(* PLC project lng-production, Generated TextualNotationConverter 1.0 *)
(* stored: creationDateTime 2025-07-30T12:00:00, modificationDateTime 2025-01-30T12:00:00 *)

FUNCTION_BLOCK ANALOG_IN
  VAR_INPUT
    Name : STRING;
    Description : STRING;
    Raw_Signal : REAL;
    PV_High : REAL;
    PV_Low : REAL;
    Scaling_Slope : REAL;
    Scaling_Offset : REAL;
    Alarm_Enable : BOOL;
  END_VAR
  VAR_OUTPUT
    PV : REAL;
    High_Alarm : BOOL;
    Low_Alarm : BOOL;
    General_Fault : BOOL;
  END_VAR

            
          
END_FUNCTION_BLOCK

FUNCTION_BLOCK RATIO_CONTROL
  VAR_INPUT
    Name : STRING;
    Description : STRING;
    Auto : BOOL;
    PrimaryPV : REAL;
    SecondaryPV : REAL;
    RatioSP : REAL;
    Bias : REAL;
    TrimKp : REAL;
    TrimTi : STRING;
    MV_MIN : REAL;
    MV_MAX : REAL;
    ManOut : REAL;
    Inhibit : BOOL;
  END_VAR
  VAR_OUTPUT
    SlaveSP : REAL;
    ActiveRatio : REAL;
    RatioErr : REAL;
  END_VAR

            
          
END_FUNCTION_BLOCK

FUNCTION_BLOCK VALVE_ELECTRIC
  VAR_INPUT
    Name : STRING;
    Description : STRING;
    Control_Signal : REAL;
    Manual_Mode : BOOL;
    Manual_Position : REAL;
    Open_Limit : REAL;
    Close_Limit : REAL;
    Timeout : STRING;
    Inhibit : BOOL;
  END_VAR
  VAR_OUTPUT
    Valve_Position : REAL;
    Feedback_Pos : REAL;
    Valve_Moving : BOOL;
    Position_Error : BOOL;
    Alarm : BOOL;
  END_VAR

            
          
END_FUNCTION_BLOCK

PROGRAM Section2
  VAR
    FT101_FeedGasFlow_PV : REAL;
    IT102_LiqSepFlow_PV : REAL;
    LT101_SlugCatcherLevel_PV : REAL;
    DP101_InletSepDP_PV : REAL;
    DP102_InletSepDP_PV : REAL;
    IIC101_LiqSepFlow_SP : REAL;
    IIC101_CalculatedRatio : REAL;
  END_VAR
  VAR
    DP-101 : ANALOG_IN;
    DP-102 : ANALOG_IN;
    FT-101 : ANALOG_IN;
    IT-102 : ANALOG_IN;
    LT-101 : ANALOG_IN;
    IIC-101 : RATIO_CONTROL;
    LCV-101 : VALVE_ELECTRIC;
  END_VAR

(* FBD diagram, written out as Structured Text *)
DP-101(PV_High := 10, PV_Low := 0, Alarm_Enable := TRUE, Scaling_Slope := 0.625, Scaling_Offset := -2.5);
DP101_InletSepDP_PV := DP-101.PV;
DP-102(PV_High := 10, PV_Low := 0, Alarm_Enable := TRUE, Scaling_Slope := 0.625, Scaling_Offset := -2.5);
DP102_InletSepDP_PV := DP-102.PV;
FT-101(PV_High := 5000, PV_Low := 100, Alarm_Enable := TRUE, Scaling_Slope := 312.5, Scaling_Offset := -1250);
FT101_FeedGasFlow_PV := FT-101.PV;
IT-102(PV_High := 2000, PV_Low := 0, Alarm_Enable := TRUE, Scaling_Slope := 125, Scaling_Offset := -500);
LT-101(PV_High := 80, PV_Low := 0, Alarm_Enable := TRUE, Scaling_Slope := 6.25, Scaling_Offset := -25);
IIC-101(PrimaryPV := FT-101.PV, SecondaryPV := IT-102.PV, Inhibit := DP-101.High_Alarm OR DP-102.High_Alarm OR LT-101.High_Alarm OR FT-101.Low_Alarm, Auto := TRUE, RatioSP := 2.5, Bias := 0, MV_MIN := 0, MV_MAX := 2000, ManOut := 500);
IIC101_CalculatedRatio := IIC-101.ActiveRatio;
IIC101_LiqSepFlow_SP := IIC-101.SlaveSP;
IT102_LiqSepFlow_PV := IT-102.PV;
LT101_SlugCatcherLevel_PV := LT-101.PV;
LCV-101(Control_Signal := IIC-101.SlaveSP, Inhibit := IT-102.High_Alarm OR IT-102.Low_Alarm OR FT-101.Low_Alarm OR IT-102.General_Fault, Manual_Mode := FALSE, Manual_Position := 0, Open_Limit := 100, Close_Limit := 0);
END_PROGRAM

FUNCTION_BLOCK BOOL_IN
  VAR_INPUT
    Name : STRING;
    Description : STRING;
    Bool_In : BOOL;
    Alarm_OnTrue : BOOL;
    Alarm_OnFalse : BOOL;
    Latch_Enable : BOOL;
    Reset_Latch : BOOL;
  END_VAR
  VAR_OUTPUT
    Bool_Out : BOOL;
    Alarm_Active : BOOL;
    Latched_Status : BOOL;
  END_VAR

            
          
END_FUNCTION_BLOCK

FUNCTION_BLOCK DIGITAL_IN
  VAR_INPUT
    Name : STRING;
    Description : STRING;
    DI_Raw : BOOL;
    DebounceTime : STRING;
    EnableAlarm : BOOL;
  END_VAR
  VAR_OUTPUT
    DI_Out : BOOL;
    Fault_State : BOOL;
  END_VAR

            
          
END_FUNCTION_BLOCK

FUNCTION_BLOCK DUTY_STANDBY
  VAR_INPUT
    Name : STRING;
    Description : STRING;
    Enable : BOOL;
    StartRequest : BOOL;
    AlternateEnable : BOOL;
    ForcePumpA : BOOL;
    ForcePumpB : BOOL;
    DutyElapsed : BOOL;
    MinRunElapsed : BOOL;
    SwitchoverDelayElapsed : BOOL;
    StartTimeoutElapsed : BOOL;
    PumpA_RunFB : BOOL;
    PumpB_RunFB : BOOL;
    PumpA_Fault : BOOL;
    PumpB_Fault : BOOL;
    Reset : BOOL;
    Inhibit : BOOL;
  END_VAR
  VAR_OUTPUT
    CmdPumpA : BOOL;
    CmdPumpB : BOOL;
    ActiveIsA : BOOL;
    SwitchedDueToDuty : BOOL;
    SwitchedDueToFailure : BOOL;
    Alarm_FailedStart_A : BOOL;
    Alarm_FailedStart_B : BOOL;
    Alarm_NoAvailablePump : BOOL;
  END_VAR

            
          
END_FUNCTION_BLOCK

FUNCTION_BLOCK MOTOR_2SPD
  VAR_INPUT
    Name : STRING;
    Description : STRING;
    Start_Cmd : BOOL;
    Stop_Cmd : BOOL;
    Speed_High_Cmd : BOOL;
    Speed_Low_Cmd : BOOL;
    Inhibit : BOOL;
  END_VAR
  VAR_OUTPUT
    Motor_Start_Out : BOOL;
    FB_Running : BOOL;
    FB_Trip : BOOL;
    FB_HighSpeed : BOOL;
    FB_LowSpeed : BOOL;
    Alarm_Speed_Error : BOOL;
  END_VAR

            
          
END_FUNCTION_BLOCK

FUNCTION_BLOCK MOTOR_ON_OFF
  VAR_INPUT
    Name : STRING;
    Description : STRING;
    Start_Cmd : BOOL;
    Stop_Cmd : BOOL;
    Start_Delay : STRING;
    MinRunTime : STRING;
    Inhibit : BOOL;
  END_VAR
  VAR_OUTPUT
    Motor_Start_Out : BOOL;
    FB_Running : BOOL;
    FB_Trip : BOOL;
    Alarm_Start_Fail : BOOL;
    Alarm_Stop_Fail : BOOL;
  END_VAR

            
          
END_FUNCTION_BLOCK

FUNCTION_BLOCK MOTOR_VSD
  VAR_INPUT
    Name : STRING;
    Description : STRING;
    Start_Cmd : BOOL;
    Stop_Cmd : BOOL;
    Speed_SP : REAL;
    Accel_Ramp : STRING;
    Decel_Ramp : STRING;
    Inhibit : BOOL;
  END_VAR
  VAR_OUTPUT
    Speed_Out : REAL;
    FB_Running : BOOL;
    FB_Fault : BOOL;
    FB_Ready : BOOL;
    FB_ActualSpeed : REAL;
    Alarm_Speed_Deviation : BOOL;
    Alarm_Comm_Fail : BOOL;
  END_VAR

            
          
END_FUNCTION_BLOCK

FUNCTION_BLOCK PID_BASIC
  VAR_INPUT
    Name : STRING;
    Description : STRING;
    AUTO : BOOL;
    PV : REAL;
    SP : REAL;
    MV_MIN : REAL;
    MV_MAX : REAL;
    X0 : REAL;
    KP : REAL;
    TR : REAL;
    TD : REAL;
    PV_High : REAL;
    PV_Low : REAL;
    Deviation_Limit : REAL;
    Inhibit : BOOL;
  END_VAR
  VAR_OUTPUT
    PV_High_Alarm : BOOL;
    PV_Low_Alarm : BOOL;
    Deviation_Alarm : BOOL;
    XOUT : REAL;
  END_VAR

            
          
END_FUNCTION_BLOCK

FUNCTION_BLOCK SPLIT_RANGE
  VAR_INPUT
    Name : STRING;
    Description : STRING;
    IN : REAL;
    Split_Point : REAL;
    Output1_Start : REAL;
    Output1_End : REAL;
    Output2_Start : REAL;
    Output2_End : REAL;
  END_VAR
  VAR_OUTPUT
    OUT1 : REAL;
    OUT2 : REAL;
  END_VAR

            
          
END_FUNCTION_BLOCK

FUNCTION_BLOCK VALVE_ON_OFF
  VAR_INPUT
    Name : STRING;
    Description : STRING;
    Open_Cmd : BOOL;
    Close_Cmd : BOOL;
    Timeout : STRING;
    Inhibit : BOOL;
  END_VAR
  VAR_OUTPUT
    FB_Opened : BOOL;
    FB_Closed : BOOL;
    Valve_Open_Out : BOOL;
    Valve_Close_Out : BOOL;
    Alarm_Position_Error : BOOL;
    Alarm_General : BOOL;
  END_VAR

            
          
END_FUNCTION_BLOCK

FUNCTION_BLOCK VOTING_ANALOG
  VAR_INPUT
    Name : STRING;
    Description : STRING;
    Input1 : REAL;
    Input2 : REAL;
    Input3 : REAL;
    Deviation_Limit : REAL;
    Voting_Scheme : STRING;
    EnableAlarm : BOOL;
    Inhibit : BOOL;
  END_VAR
  VAR_OUTPUT
    Voted_Output : REAL;
    Sensor1_Fault : BOOL;
    Sensor2_Fault : BOOL;
    Sensor3_Fault : BOOL;
    Alarm_Voting_Error : BOOL;
    Healthy_Sensors_Count : INT;
  END_VAR

            
          
END_FUNCTION_BLOCK

PROGRAM Section3
  VAR
    TT201_Temperature_PV : REAL;
    TIC201_Output_MV_Pct : REAL;
    PT201_Pressure_PV : REAL;
    LT201_Level_PV : REAL;
    AI201_CO2_PV : REAL;
  END_VAR
  VAR
    AI-201 : ANALOG_IN;
    FV-101 : VALVE_ELECTRIC;
    LT-201 : ANALOG_IN;
    PT-201 : ANALOG_IN;
    TIC-201 : PID_BASIC;
    TT-201 : ANALOG_IN;
  END_VAR
  VAR  (* added by the conversion: wires and edge detectors of the diagram *)
    _OR56_OUT : BOOL;
  END_VAR

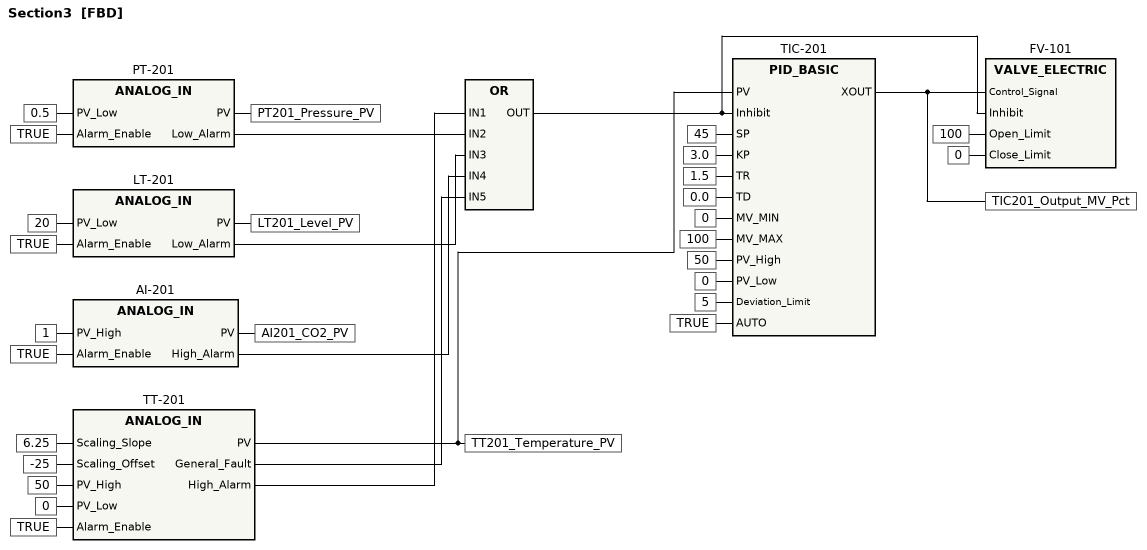
(* FBD diagram, written out as Structured Text *)
AI-201(PV_High := 1, Alarm_Enable := TRUE);
AI201_CO2_PV := AI-201.PV;
LT-201(PV_Low := 20, Alarm_Enable := TRUE);
LT201_Level_PV := LT-201.PV;
PT-201(PV_Low := 0.5, Alarm_Enable := TRUE);
PT201_Pressure_PV := PT-201.PV;
TT-201(Scaling_Slope := 6.25, Scaling_Offset := -25, PV_High := 50, PV_Low := 0, Alarm_Enable := TRUE);
_OR56_OUT := TT-201.High_Alarm OR PT-201.Low_Alarm OR LT-201.Low_Alarm OR AI-201.High_Alarm OR TT-201.General_Fault;
TIC-201(PV := TT-201.PV, Inhibit := _OR56_OUT, SP := 45, KP := 3.0, TR := 1.5, TD := 0.0, MV_MIN := 0, MV_MAX := 100, PV_High := 50, PV_Low := 0, Deviation_Limit := 5, AUTO := TRUE);
TIC201_Output_MV_Pct := TIC-201.XOUT;
TT201_Temperature_PV := TT-201.PV;
FV-101(Control_Signal := TIC-201.XOUT, Inhibit := _OR56_OUT, Open_Limit := 100, Close_Limit := 0);
END_PROGRAM

PROGRAM Section4
  VAR
    FT301_FeedGasFlow_PV : REAL;
    AI302_Mercury_PV : REAL;
    AI303_Mercury_PV : REAL;
    AI304_OutletH2O_PV : REAL;
    DP301_BedDP_PV : REAL;
    FFIC303_RegenGasFlow_SP : REAL;
  END_VAR
  VAR
    AI-302 : ANALOG_IN;
    AI-303 : ANALOG_IN;
    AI-304 : ANALOG_IN;
    DI-301 : DIGITAL_IN;
    DP-301 : ANALOG_IN;
    FIC-302 : PID_BASIC;
    FT-301 : ANALOG_IN;
    FV-302 : VALVE_ELECTRIC;
    FFIC-303 : RATIO_CONTROL;
  END_VAR
  VAR  (* added by the conversion: wires and edge detectors of the diagram *)
    _OR91_OUT : BOOL;
  END_VAR

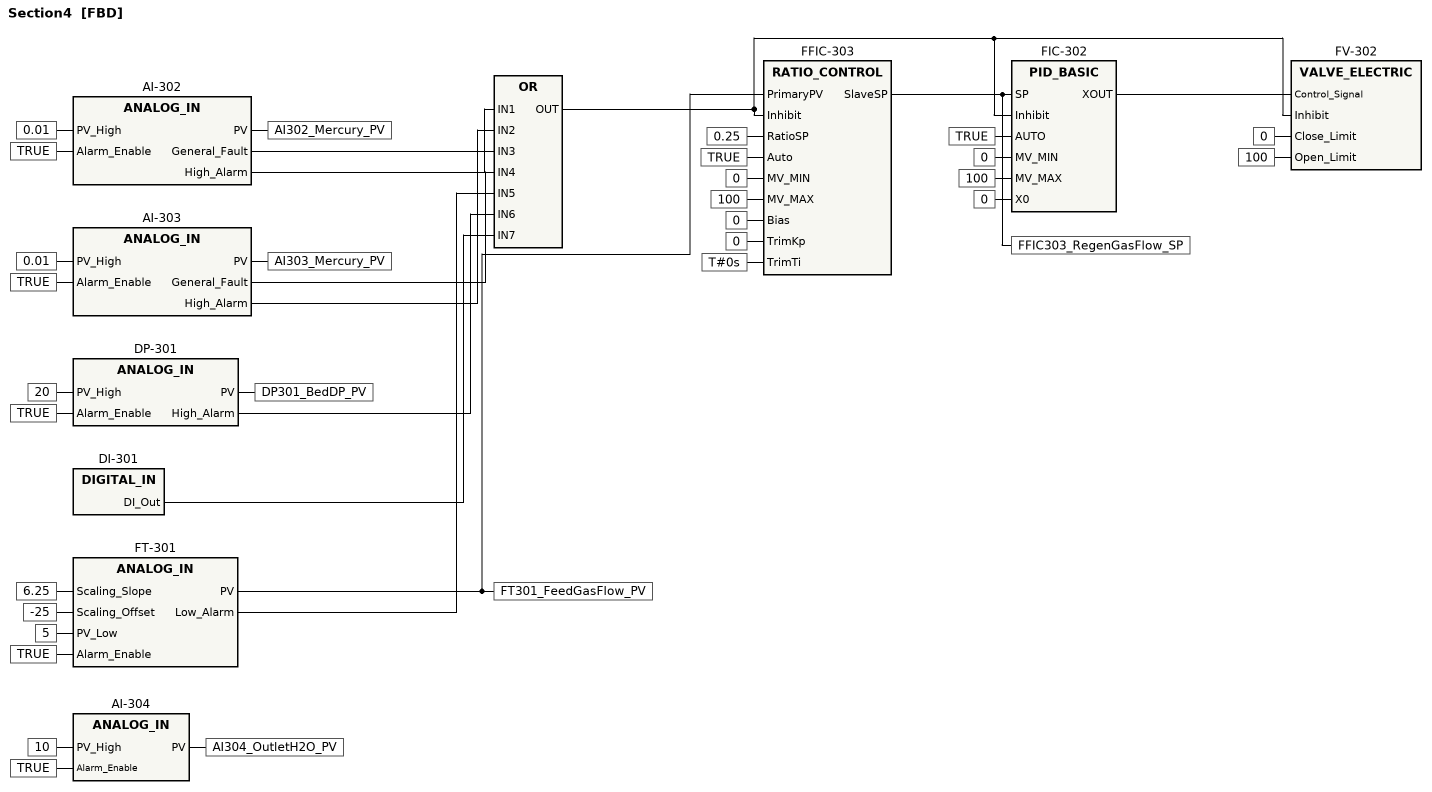
(* FBD diagram, written out as Structured Text *)
AI-302(PV_High := 0.01, Alarm_Enable := TRUE);
AI302_Mercury_PV := AI-302.PV;
AI-303(PV_High := 0.01, Alarm_Enable := TRUE);
AI303_Mercury_PV := AI-303.PV;
AI-304(PV_High := 10, Alarm_Enable := TRUE);
AI304_OutletH2O_PV := AI-304.PV;
DP-301(PV_High := 20, Alarm_Enable := TRUE);
DP301_BedDP_PV := DP-301.PV;
FT-301(Scaling_Slope := 6.25, Scaling_Offset := -25, PV_Low := 5, Alarm_Enable := TRUE);
DI-301();
_OR91_OUT := AI-302.High_Alarm OR AI-303.High_Alarm OR AI-302.General_Fault OR AI-303.General_Fault OR FT-301.Low_Alarm OR DP-301.High_Alarm OR DI-301.DI_Out;
FFIC-303(PrimaryPV := FT-301.PV, Inhibit := _OR91_OUT, RatioSP := 0.25, Auto := TRUE, MV_MIN := 0, MV_MAX := 100, Bias := 0, TrimKp := 0, TrimTi := T#0s);
FFIC303_RegenGasFlow_SP := FFIC-303.SlaveSP;
FT301_FeedGasFlow_PV := FT-301.PV;
FIC-302(SP := FFIC-303.SlaveSP, Inhibit := _OR91_OUT, AUTO := TRUE, MV_MIN := 0, MV_MAX := 100, X0 := 0);
FV-302(Control_Signal := FIC-302.XOUT, Inhibit := _OR91_OUT, Close_Limit := 0, Open_Limit := 100);
END_PROGRAM

PROGRAM Section5
  VAR
    PT_401_Pressure_PV : REAL;
    PT_401A_Pressure_PV : REAL;
    PT_401B_Pressure_PV : REAL;
    PT_401C_Pressure_PV : REAL;
    TT_105_Temperature_PV : REAL;
    TT_106_Temperature_PV : REAL;
    TT_107_Temperature_PV : REAL;
    FA_401_Flow_PV : REAL;
    FA_402A_Flow_PV : REAL;
    FA_402B_Flow_PV : REAL;
    FA_402C_Flow_PV : REAL;
    PVT_401_VotedPressure : REAL;
    TVT_402_VotedTemperature : REAL;
    PVT_401_Healthy_Count : INT;
    DA_401A_Deviation : BOOL;
    DA_401B_Deviation : BOOL;
    DA_401C_Deviation : BOOL;
    DA_402A_Deviation : BOOL;
    DA_402B_Deviation : BOOL;
    DA_402C_Deviation : BOOL;
    DA_402_Degraded : BOOL;
    MA_401_Alarm : BOOL;
  END_VAR
  VAR
    PT-401 : ANALOG_IN;
    PT-401A : ANALOG_IN;
    PT-401B : ANALOG_IN;
    PT-401C : ANALOG_IN;
    TT-105 : ANALOG_IN;
    TT-106 : ANALOG_IN;
    TT-107 : ANALOG_IN;
    FA-401 : ANALOG_IN;
    FA-402A : ANALOG_IN;
    FA-402B : ANALOG_IN;
    FA-402C : ANALOG_IN;
    PVT-401 : VOTING_ANALOG;
    TVT-402 : VOTING_ANALOG;
    PV-102_Control : PID_BASIC;
    PV-102 : VALVE_ELECTRIC;
    FV-107 : VALVE_ELECTRIC;
    XV-104 : VALVE_ON_OFF;
  END_VAR
  VAR  (* added by the conversion: wires and edge detectors of the diagram *)
    _MULT134_OUT : REAL;
    _OR155_OUT : BOOL;
    _AND132_OUT : BOOL;
    _OR156_OUT : BOOL;
  END_VAR

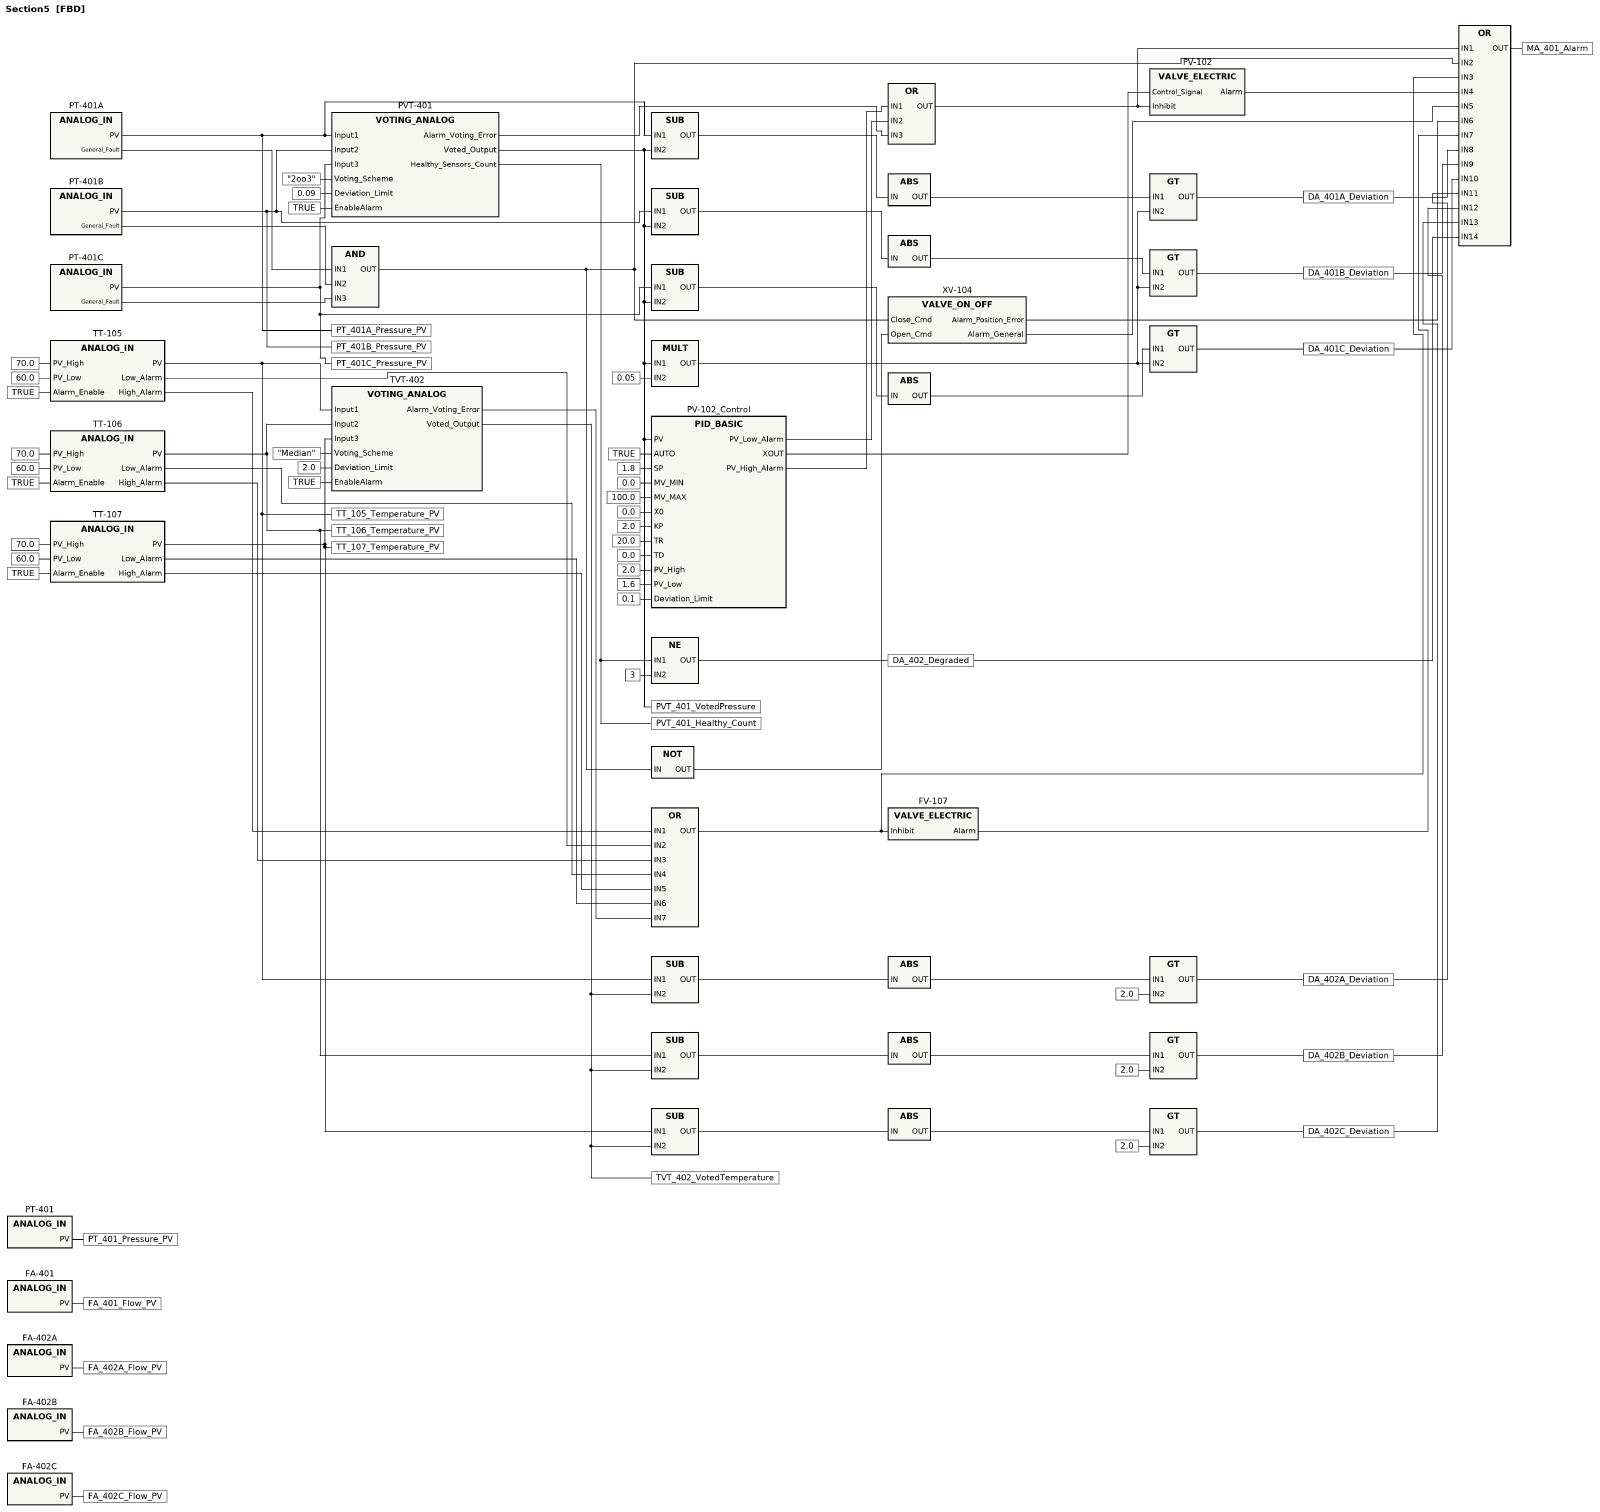
(* FBD diagram, written out as Structured Text *)
PT-401A();
PT-401B();
PT-401C();
PVT-401(Input1 := PT-401A.PV, Input2 := PT-401B.PV, Input3 := PT-401C.PV, Voting_Scheme := "2oo3", Deviation_Limit := 0.09, EnableAlarm := TRUE);
_MULT134_OUT := MULT(PVT-401.Voted_Output, 0.05);
DA_401A_Deviation := ABS(PT-401A.PV - PVT-401.Voted_Output) > _MULT134_OUT;
DA_401B_Deviation := ABS(PT-401B.PV - PVT-401.Voted_Output) > _MULT134_OUT;
DA_401C_Deviation := ABS(PT-401C.PV - PVT-401.Voted_Output) > _MULT134_OUT;
TT-105(PV_High := 70.0, PV_Low := 60.0, Alarm_Enable := TRUE);
TT-106(PV_High := 70.0, PV_Low := 60.0, Alarm_Enable := TRUE);
TT-107(PV_High := 70.0, PV_Low := 60.0, Alarm_Enable := TRUE);
TVT-402(Input1 := TT-105.PV, Input2 := TT-106.PV, Input3 := TT-107.PV, Voting_Scheme := "Median", Deviation_Limit := 2.0, EnableAlarm := TRUE);
DA_402A_Deviation := ABS(TT-105.PV - TVT-402.Voted_Output) > 2.0;
DA_402B_Deviation := ABS(TT-106.PV - TVT-402.Voted_Output) > 2.0;
DA_402C_Deviation := ABS(TT-107.PV - TVT-402.Voted_Output) > 2.0;
DA_402_Degraded := PVT-401.Healthy_Sensors_Count <> 3;
FA-401();
FA_401_Flow_PV := FA-401.PV;
FA-402A();
FA_402A_Flow_PV := FA-402A.PV;
FA-402B();
FA_402B_Flow_PV := FA-402B.PV;
FA-402C();
FA_402C_Flow_PV := FA-402C.PV;
PV-102_Control(PV := PVT-401.Voted_Output, AUTO := TRUE, SP := 1.8, MV_MIN := 0.0, MV_MAX := 100.0, X0 := 0.0, KP := 2.0, TR := 20.0, TD := 0.0, PV_High := 2.0, PV_Low := 1.6, Deviation_Limit := 0.1);
_OR155_OUT := PV-102_Control.PV_High_Alarm OR PV-102_Control.PV_Low_Alarm OR PVT-401.Alarm_Voting_Error;
_AND132_OUT := PT-401A.General_Fault AND PT-401B.General_Fault AND PT-401C.General_Fault;
_OR156_OUT := TT-105.High_Alarm OR TT-105.Low_Alarm OR TT-106.High_Alarm OR TT-106.Low_Alarm OR TT-107.High_Alarm OR TT-107.Low_Alarm OR TVT-402.Alarm_Voting_Error;
PV-102(Control_Signal := PV-102_Control.XOUT, Inhibit := _OR155_OUT);
XV-104(Close_Cmd := _AND132_OUT, Open_Cmd := NOT _AND132_OUT);
FV-107(Inhibit := _OR156_OUT);
MA_401_Alarm := _OR155_OUT OR _AND132_OUT OR _OR156_OUT OR PV-102.Alarm OR XV-104.Alarm_General OR XV-104.Alarm_Position_Error OR FV-107.Alarm OR ABS(PT-401A.PV - PVT-401.Voted_Output) > _MULT134_OUT OR ABS(PT-401B.PV - PVT-401.Voted_Output) > _MULT134_OUT OR ABS(PT-401C.PV - PVT-401.Voted_Output) > _MULT134_OUT OR ABS(TT-105.PV - TVT-402.Voted_Output) > 2.0 OR ABS(TT-106.PV - TVT-402.Voted_Output) > 2.0 OR ABS(TT-107.PV - TVT-402.Voted_Output) > 2.0 OR PVT-401.Healthy_Sensors_Count <> 3;
PT_401A_Pressure_PV := PT-401A.PV;
PT_401B_Pressure_PV := PT-401B.PV;
PT_401C_Pressure_PV := PT-401C.PV;
PT-401();
PT_401_Pressure_PV := PT-401.PV;
PVT_401_Healthy_Count := PVT-401.Healthy_Sensors_Count;
PVT_401_VotedPressure := PVT-401.Voted_Output;
TT_105_Temperature_PV := TT-105.PV;
TT_106_Temperature_PV := TT-106.PV;
TT_107_Temperature_PV := TT-107.PV;
TVT_402_VotedTemperature := TVT-402.Voted_Output;
END_PROGRAM

PROGRAM Section6
  VAR
    FT_501_PropaneFlow_PV : REAL;
    FT_502_MRFlow_PV : REAL;
    PT_501_Pressure_PV : REAL;
    TIT_102_Temperature_PV : REAL;
    FIC_504_SP_Selected : REAL;
    FFIC_503_ActiveRatio : REAL;
    FV_502_ControlSignal : REAL;
    FV_501_Feedback_Pos : REAL;
    RatioBias_Manual : REAL;
    AntiSurgeActive : BOOL;
    PropaneLowFlow : BOOL;
    FlowRangeOrFault : BOOL;
    RatioControlInhibit : BOOL;
    RatioDevHigh_ALM : BOOL;
    RatioDevLow_ALM : BOOL;
  END_VAR
  VAR
    FT-501 : ANALOG_IN;
    FT-502 : ANALOG_IN;
    PT-501 : ANALOG_IN;
    TIT-102 : ANALOG_IN;
    FFIC-503 : RATIO_CONTROL;
    FIC-504 : PID_BASIC;
    FV-502 : VALVE_ELECTRIC;
    FV-501 : VALVE_ELECTRIC;
  END_VAR
  VAR  (* added by the conversion: wires and edge detectors of the diagram *)
    _OR233_OUT : BOOL;
    _LT237_OUT : BOOL;
    _TON236_OUT : BOOL;
    _OR234_OUT : BOOL;
    _SEL240_OUT : REAL;
  END_VAR

(* FBD diagram, written out as Structured Text *)
FT-501(Scaling_Slope := 312.5, Scaling_Offset := -1250.0, Alarm_Enable := TRUE, PV_High := 5000.0, PV_Low := 500.0);
FT-502(Scaling_Slope := 125.0, Scaling_Offset := -500.0, Alarm_Enable := TRUE, PV_High := 2000.0, PV_Low := 200.0);
TIT-102(Scaling_Slope := 12.5, Scaling_Offset := -250.0, Alarm_Enable := TRUE, PV_High := -155.0);
_OR233_OUT := FT-501.High_Alarm OR FT-501.Low_Alarm OR FT-502.High_Alarm OR FT-502.Low_Alarm OR FT-501.General_Fault OR FT-502.General_Fault;
_LT237_OUT := FT-501.PV < 500.0;
FV-501(Manual_Mode := TRUE, Manual_Position := 0.0, Open_Limit := 100.0, Close_Limit := 0.0, Timeout := T#30s);
_TON236_OUT := TON(FV-501.Feedback_Pos >= 99.0, T#5s);
PT-501(Scaling_Slope := 0.1875, Scaling_Offset := -0.75, Alarm_Enable := TRUE, PV_Low := 2.0);
_OR234_OUT := _OR233_OUT OR _LT237_OUT OR _TON236_OUT OR PT-501.Low_Alarm;
FFIC-503(PrimaryPV := FT-501.PV, SecondaryPV := FT-502.PV, MV_MIN := FT-501.PV / 3.0, MV_MAX := FT-501.PV / 2.0, RatioSP := SEL(TIT-102.High_Alarm, 0.0, 0.1) + 0.4 + RatioBias_Manual, Inhibit := _OR234_OUT, Auto := NOT _OR234_OUT, Bias := 0.0, TrimKp := 0.0, TrimTi := T#0s);
FFIC_503_ActiveRatio := FFIC-503.ActiveRatio;
_SEL240_OUT := SEL(SEL(SEL(_TON236_OUT, FFIC-503.SlaveSP, 1000.0), _LT237_OUT, 100.0), _OR233_OUT, 500.0);
FIC_504_SP_Selected := _SEL240_OUT;
FT_501_PropaneFlow_PV := FT-501.PV;
FT_502_MRFlow_PV := FT-502.PV;
FV_501_Feedback_Pos := FV-501.Feedback_Pos;
FIC-504(SP := _SEL240_OUT, Inhibit := _OR234_OUT, PV := FT-502.PV, AUTO := TRUE, MV_MIN := 0.0, MV_MAX := 100.0, KP := 1.5, TR := 30.0, TD := 0.0, PV_High := 2000.0, PV_Low := 200.0, Deviation_Limit := 100.0);
FV_502_ControlSignal := FIC-504.XOUT;
PT_501_Pressure_PV := PT-501.PV;
RatioDevHigh_ALM := TON(FFIC-503.RatioErr > 0.2, T#10s);
RatioDevLow_ALM := TON(FFIC-503.RatioErr < (-0.2), T#10s);
TIT_102_Temperature_PV := TIT-102.PV;
FV-502(Inhibit := _OR234_OUT, Control_Signal := FIC-504.XOUT, Manual_Mode := FALSE, Manual_Position := 0.0, Open_Limit := 100.0, Close_Limit := 0.0, Timeout := T#30s);
END_PROGRAM

PROGRAM Section7
  VAR
    FT-601A_LNGFlow_PV : REAL;
    FT-601B_BOGFlow_PV : REAL;
    LIT-601_TankLevel_PV : REAL;
    FT-601B_SP_FromRatio : REAL;
    FFIC-601_RatioDeviation : REAL;
  END_VAR
  VAR
    FT-601A : ANALOG_IN;
    FT-601B : ANALOG_IN;
    LIT-601 : ANALOG_IN;
    LT-601 : ANALOG_IN;
    FFIC-601 : RATIO_CONTROL;
    FIC-601B : PID_BASIC;
    FV-601B : VALVE_ELECTRIC;
    C-601 : MOTOR_ON_OFF;
    HS-601 : DIGITAL_IN;
  END_VAR

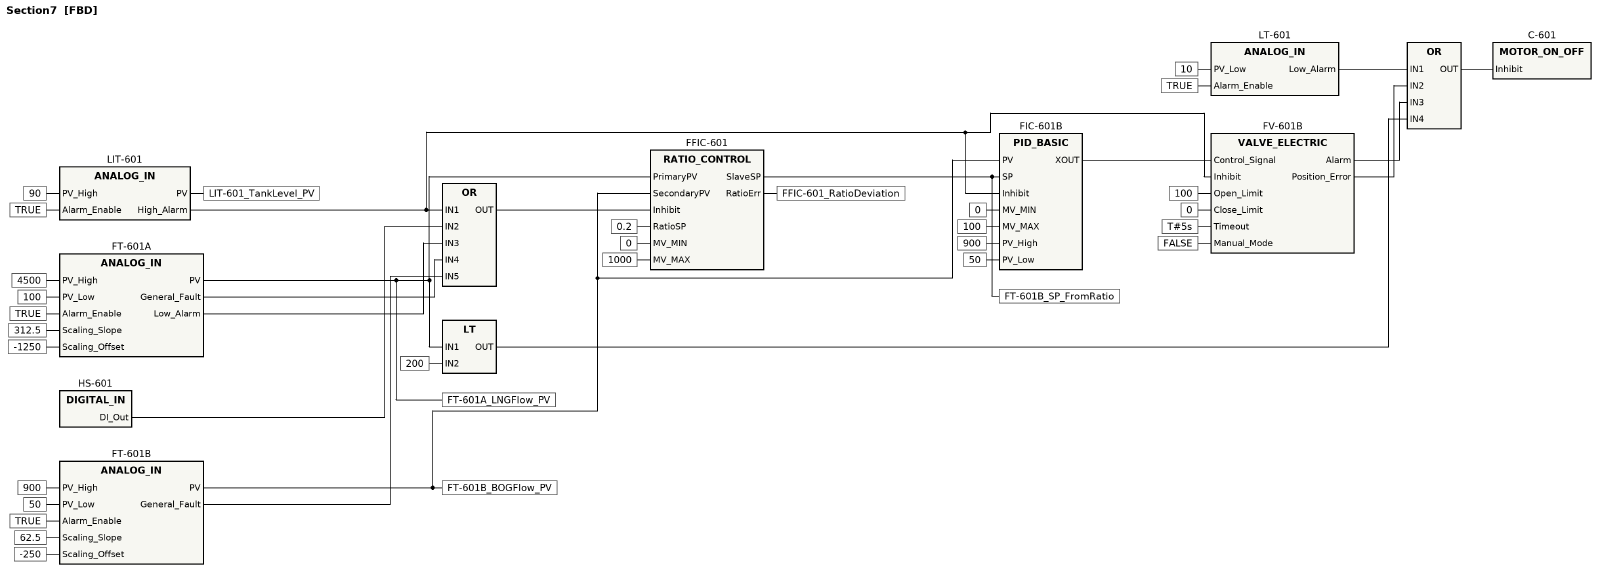
(* FBD diagram, written out as Structured Text *)
FT-601A(PV_High := 4500, PV_Low := 100, Alarm_Enable := TRUE, Scaling_Slope := 312.5, Scaling_Offset := -1250);
FT-601B(PV_High := 900, PV_Low := 50, Alarm_Enable := TRUE, Scaling_Slope := 62.5, Scaling_Offset := -250);
LIT-601(PV_High := 90, Alarm_Enable := TRUE);
HS-601();
FFIC-601(PrimaryPV := FT-601A.PV, SecondaryPV := FT-601B.PV, Inhibit := LIT-601.High_Alarm OR HS-601.DI_Out OR FT-601A.Low_Alarm OR FT-601A.General_Fault OR FT-601B.General_Fault, RatioSP := 0.2, MV_MIN := 0, MV_MAX := 1000);
FFIC-601_RatioDeviation := FFIC-601.RatioErr;
FT-601A_LNGFlow_PV := FT-601A.PV;
FT-601B_BOGFlow_PV := FT-601B.PV;
FT-601B_SP_FromRatio := FFIC-601.SlaveSP;
LIT-601_TankLevel_PV := LIT-601.PV;
LT-601(PV_Low := 10, Alarm_Enable := TRUE);
FIC-601B(PV := FT-601B.PV, SP := FFIC-601.SlaveSP, Inhibit := LIT-601.High_Alarm, MV_MIN := 0, MV_MAX := 100, PV_High := 900, PV_Low := 50);
FV-601B(Control_Signal := FIC-601B.XOUT, Inhibit := LIT-601.High_Alarm, Open_Limit := 100, Close_Limit := 0, Timeout := T#5s, Manual_Mode := FALSE);
C-601(Inhibit := LT-601.Low_Alarm OR FV-601B.Position_Error OR FV-601B.Alarm OR FT-601A.PV < 200);
END_PROGRAM

CONFIGURATION Config0
  RESOURCE Res0 ON PLC
    TASK task0(INTERVAL := T#20ms, PRIORITY := 0);
    PROGRAM instance0 WITH task0 : Section2;
    PROGRAM instance_1 WITH task0 : Section3;
    PROGRAM instance_2 WITH task0 : Section4;
    PROGRAM instance_3 WITH task0 : Section5;
    PROGRAM instance_4 WITH task0 : Section6;
    PROGRAM instance_5 WITH task0 : Section7;
  END_RESOURCE
END_CONFIGURATION
